FUNCTION F_IsAtPositionCartesian : BOOL
VAR_INPUT
  actual : ST_CartesianPoint;
  target : ST_CartesianPoint;
  delta : ST_CartesianPoint;
END_VAR

F_IsAtPositionCartesian :=
  (ABS(actual.x - target.x) < delta.x)
    AND (ABS(actual.x - target.x) < delta.x)
    AND (ABS(actual.y - target.y) < delta.y)
    AND (ABS(actual.z - target.z) < delta.z)
    AND (ABS(actual.a - target.a) < delta.a)
    AND (ABS(actual.b - target.b) < delta.b)
    AND (ABS(actual.c - target.c) < delta.c);

END_FUNCTION

(* stored: Version 1.1.0.1
   POU F_IsAtPositionCartesian: Id {1229cfe9-c8b7-493f-ad8d-c311de47c79c}, SpecialFunc None *)
